{attribute 'GeneratedUsingTerminal: EL5151-0080-0016'}
{attribute addProperty BoxType "EL5151-0080-0016"}
{attribute addProperty Id "Enable_latch_CAT %Q*BOOL1Enable_latch_extern_on_positive_edgeAT %Q*BOOL1Set_counterAT %Q*BOOL1Enable_latch_extern_on_negative_edgeAT %Q*BOOL1Set_counter_valueAT %Q*UINT2"}
{attribute addProperty CRC "1876805225"}
{attribute addProperty Size "6"}
TYPE ENC_Outputs_6FDDC669 :
STRUCT
	{attribute addProperty Name "Enable_latch_C"}
	Enable_latch_C AT %Q* : BOOL;
	{attribute addProperty Name "Enable_latch_extern_on_positive_edge"}
	Enable_latch_extern_on_positive_edge AT %Q* : BOOL;
	{attribute addProperty Name "Set_counter"}
	Set_counter AT %Q* : BOOL;
	{attribute addProperty Name "Enable_latch_extern_on_negative_edge"}
	Enable_latch_extern_on_negative_edge AT %Q* : BOOL;
	{attribute addProperty Name "Set_counter_value"}
	Set_counter_value AT %Q* : UINT;
END_STRUCT
END_TYPE

(* stored: Version 1.2.0.0, ProductVersion 3.1.4024.9
   DUT ENC_Outputs_6FDDC669: Id {6457d22a-9e2c-4556-b6e8-1eade1753e33} *)
